// TIA Portal V17 export
VBScript "Codex_VBFunction_Loop"  Type=Sub, Comment="Codex VBS import/export loop test. Object name and Sub name must match."
  ' Codex closed-loop import/export verification.
  ' Keep the object name and the generated Sub name identical: Codex_VBFunction_Loop.
  SmartTags("Codex_VBS_Input") = "IN_OK"
  SmartTags("Codex_VBS_Output") = "OUT_OK"
